PROGRAM MAIN
VAR
    _tcoDriveSimpleTestContext : TcoDriveSimpleTestContext;
    _wpfContext : WpfContext;
    _wpfContextCall : BOOL := FALSE;
END_VAR

_tcoDriveSimpleTestContext.ProbeRun();

//IF _wpfContextCall THEN
	_wpfContext.Run();
//END_IF

END_PROGRAM

(* stored: Version 1.1.0.1, ProductVersion 3.1.4024.12
   POU MAIN: Id {6dac1541-74ba-49c0-be18-0d7d17fb8228}, SpecialFunc None *)
